FUNCTION_BLOCK Stage9 (* Template for a Basic Function Block Type *)
  (* Standard: 61499-2 *)
  (* Version 1.0, 2021-06-20, HP *)
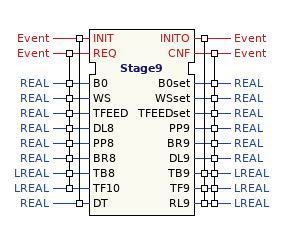
  EVENT_INPUT
    INIT WITH DT; (* Initialization Request *)
    REQ WITH B0, WS, TFEED, DL8, PP8, BR8, TB8, TF10; (* Normal Execution Request *)
  END_EVENT
  EVENT_OUTPUT
    INITO WITH TB9, TF9, RL9; (* Initialization Confirm *)
    CNF WITH TB9, DL9, TF9, BR9, PP9, TFEEDset, WSset, B0set, RL9; (* Execution Confirmation *)
  END_EVENT
  VAR_INPUT
    B0 : REAL;
    WS : REAL;
    TFEED : REAL;
    DL8 : REAL;
    PP8 : REAL;
    BR8 : REAL;
    TB8 : LREAL;
    TF10 : LREAL;
    DT : REAL;
  END_VAR
  VAR_OUTPUT
    B0set : REAL;
    WSset : REAL;
    TFEEDset : REAL;
    PP9 : REAL;
    BR9 : REAL;
    DL9 : REAL;
    TB9 : LREAL;
    TF9 : LREAL;
    RL9 : LREAL;
  END_VAR
  VAR
    AB : REAL; (* internal variabel *)
    UU : REAL;
    TREF : REAL;
    AD : REAL;
    AHC : REAL;
    AHR : REAL;
    AS : REAL;
    REC : REAL;
    WN : REAL;
    WN_1 : REAL;
    XKN : REAL;
    C1 : REAL;
    HS : REAL;
    G : REAL;
    W1 : REAL;
    TFREC : REAL;
    TS : REAL;
    DTS : REAL;
    TF9_last : REAL;
    RL9_last : REAL;
    TB9_last : REAL;
    USS : REAL;
    RHOB : REAL;
    CPB : REAL;
    CPF : REAL;
    FMW : REAL;
    HLV : REAL;
    HV : REAL;
    BPR : REAL;
    FMC : REAL;
    U : REAL;
    A : REAL;
    B : REAL;
    C : REAL;
    D1 : REAL;
    d : REAL;
    a : REAL;
    A1 : REAL;
    A2 : REAL;
    A3 : REAL;
    A4 : REAL;
    A5 : REAL;
    A6 : REAL;
    p : REAL;
    q : REAL;
    TC : REAL;
    PC : REAL;
    DTB9 : REAL;
    DEN9 : REAL;
    DH9 : REAL;
    DP9 : REAL;
    DPDH9 : REAL;
    DT9 : REAL;
    m : REAL;
    n : REAL;
    VR9 : REAL;
    DELTA9 : REAL;
    DELTA31 : REAL;
    DELTA53 : REAL;
    DELTA9_last : REAL;
    DELTA31_last : REAL;
    DELTA53_last : REAL;
  END_VAR
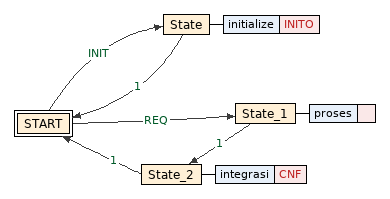
  EC_STATES
    START; (* Initial State *)
    State : initialize -> INITO;
    State_1 : proses;
    State_2 : integrasi -> CNF;
  END_STATES
  EC_TRANSITIONS
    START TO State := INIT;
    State TO START := 1;
    START TO State_1 := REQ;
    State_1 TO State_2 := 1;
    State_2 TO START := 1;
  END_TRANSITIONS
  ALGORITHM initialize IN ST: (* Initialization algorithm *)
TREF :=273.15;
AB :=57.2727;
AHC :=4069.2;
AHR :=2639.7;
AS :=3225.7;
REC :=0.0;
//TF2:=TF2;

//TFEED :=TFEED1+TREF;
 //TS:=TS1+TREF;
WN :=3.0;
XKN :=0.68;
HS:=0.11;
G :=9.81;
W1 :=0.50;

RL9 := 0.565913411730399;
TB9 := 343.141074721262;
TF9 := 339.272674118834;
TF10 := 336.687818219045;


RL9_last :=RL9;
TB9_last :=TB9;
TF9_last :=TF9;
  END_ALGORITHM
  ALGORITHM proses IN ST: (* kalkulasi *)
UU := TFEED;
U :=UU;

USS :=49.767;
C1 :=0.625;
RHOB :=1032.4; //maassa jenis brine
CPB :=1.00; //heatcapacity Brine
CPF :=1.00; //heat capacity feed
FMW :=23654.0;
HLV :=563.7959;
HV :=625.1971;
BPR :=2.192;
FMC :=34736.09;
//U :=UU; //feed temp



///  Calculate the physical properties

//A :=3.2437814;
//B :=5.86826*0.001;
//C :=1.1702379*0.00000001;
//D1 :=2.1878462*0.001;
//TC :=647.27;
//PC :=218.167;


A1 :=3.2437814;
A2:=5.86826*0.001;
A3:=1.1702379*0.00000001;
A4 :=2.1878462*0.001;
A5 :=647.27;
A6 :=218.167;

DTB9 :=A5-TB9;
DEN9 :=(A1+A2*DTB9+A3*DTB9*DTB9*DTB9)/(1+A4*DTB9)*DTB9/TB9;
p:=DEN9;
q:=10.0;
PP9 :=A6/(EXPT(q, p));

// calculate the brine flow rates
DP9:=PP8-PP9;
DH9:=RL9-C1*HS;
DPDH9 :=DP9*101000+G*RHOB*DH9;
m:=DPDH9*RHOB;
n:=0.5;
BR9 :=WN*XKN*RL9*(EXPT(m, n));
BR9 :=BR9*60.0/1000.0;

// calculate the vapor flow rates

DT9 :=TB9-BPR/1.8-(TF10+TF9)*0.5;
VR9 :=U*AHC*DT9/HLV/1000.0;
DL9 :=DL8+VR9;


//// state equation
DELTA9 :=(BR8-BR9-VR9)*1000.0/RHOB/AB;
DELTA31 :=((BR8*CPB*(TB8-TB9))-VR9*(HV-CPB*(TB9-TREF)))*1000.0/AB/RHOB/CPB/RL9;
DELTA53 :=(B0*CPF*(TF10-TF9)*1000+(U*AHC*DT9))/FMW/CPF;
  END_ALGORITHM
  ALGORITHM integrasi IN ST: (* new algorithm *)
B0set:=B0;
WSset:=WS ;
TFEEDset:=TFEED;
//integrasi
RL9 := (DELTA9 + DELTA9_last)*0.5*DT + RL9_last;
DELTA9_last :=DELTA9 ;
RL9_last :=RL9;

TB9:= (DELTA31 + DELTA31_last)*0.5*DT + TB9_last;
DELTA31_last :=DELTA31 ;
TB9_last:=TB9;

TF9 := (DELTA53 + DELTA53_last)*0.5*DT + TF9_last;
DELTA53_last :=DELTA53 ;
TF9_last :=TF9;
  END_ALGORITHM
END_FUNCTION_BLOCK
